% RSLogix 500 project AUTOGENE.RSS, saved by version 8.30.00.16 %
PROJECT "AUTOGENE"    % processor: Bul.1763 MicroLogix 1100 Series B %

PROGRAM FILES
  LAD 2 "MAIN"  4 rungs
  LAD 3 "DIG INPUT"  7 rungs
  LAD 5 "CONTROLS"  6 rungs
  LAD 6 "ALARMS"  12 rungs

DATA FILES
  O0 OUTPUT  6 elements
  I1 INPUT  12 elements
  S2 STATUS  66 elements
  B3 BINARY  4 elements
  T4 TIMER  3 elements
  C5 COUNTER  1 elements
  R6 CONTROL  1 elements
  N7 INTEGER  2 elements
  F8 FLOAT  1 elements

LADDER 2 "MAIN"
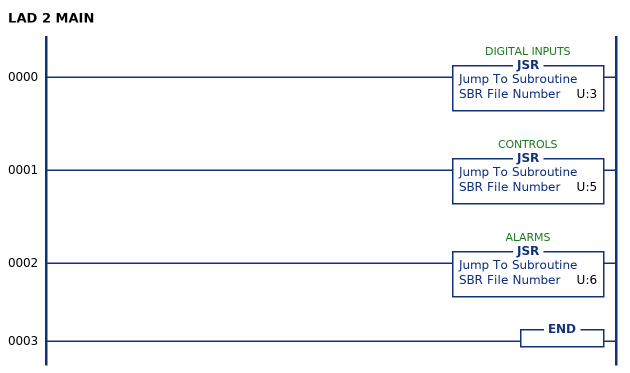
% Rung: 0 %
SOR JSR U:3 EOR
%   U:3  "DIGITAL INPUTS" %
% Rung: 1 %
SOR JSR U:5 EOR
%   U:5  "CONTROLS" %
% Rung: 2 %
SOR JSR U:6 EOR
%   U:6  "ALARMS" %
% Rung: 3 %
SOR END EOR

LADDER 3 "DIG INPUT"
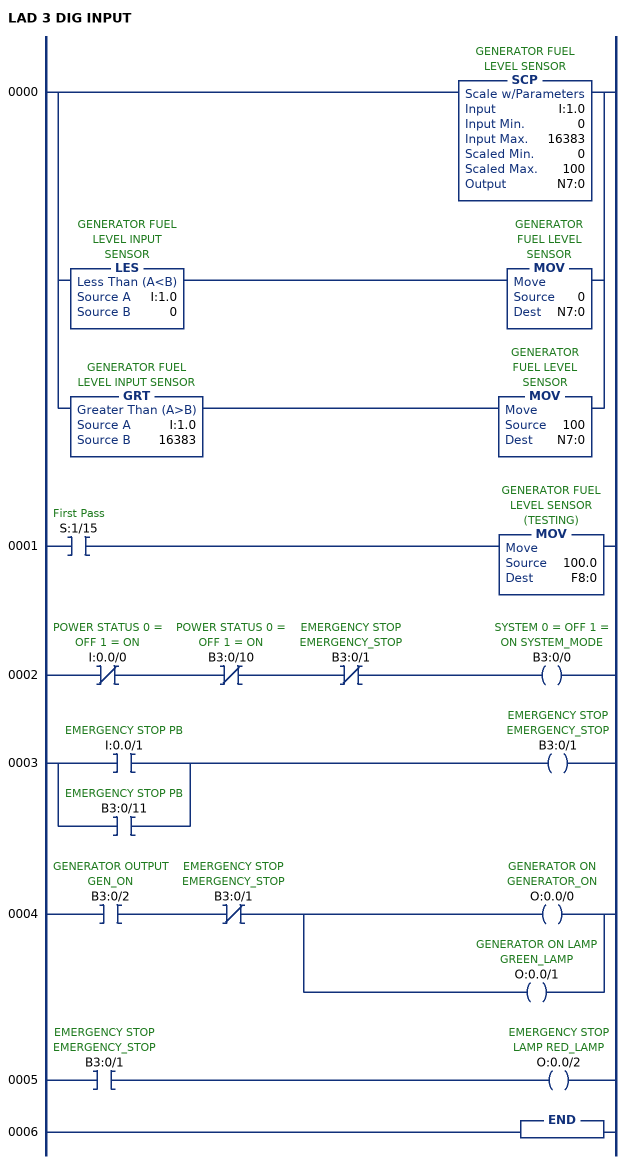
% Rung: 0 %
SOR BST SCP I:1.0 0 16383 0 100 N7:0 NXB LES I:1.0 0 MOV 0 N7:0 NXB GRT I:1.0 16383 MOV 100 N7:0 BND EOR
%   I:1.0  "GENERATOR FUEL LEVEL INPUT SENSOR" %
%   N7:0  "GENERATOR FUEL LEVEL SENSOR" %
% Rung: 1 %
SOR XIC S:1/15 MOV 100.0 F8:0 EOR
%   S:1/15  "First Pass" %
%   F8:0  "GENERATOR FUEL LEVEL SENSOR (TESTING)" %
% Rung: 2 %
SOR XIO I:0.0/0 XIO B3:0/10 XIO B3:0/1 OTE B3:0/0 EOR
%   I:0.0/0  "POWER STATUS 0 = OFF 1 = ON" %
%   B3:0/10  "POWER STATUS 0 = OFF 1 = ON" %
%   B3:0/1  EMERGENCY_STOP  "EMERGENCY STOP" %
%   B3:0/0  SYSTEM_MODE  "SYSTEM 0 = OFF 1 = ON" %
% Rung: 3 %
SOR BST XIC I:0.0/1 NXB XIC B3:0/11 BND OTE B3:0/1 EOR
%   I:0.0/1  "EMERGENCY STOP PB" %
%   B3:0/11  "EMERGENCY STOP PB" %
%   B3:0/1  EMERGENCY_STOP  "EMERGENCY STOP" %
% Rung: 4 %
SOR XIC B3:0/2 XIO B3:0/1 BST OTE O:0.0/0 NXB OTE O:0.0/1 BND EOR
%   B3:0/2  GEN_ON  "GENERATOR OUTPUT" %
%   B3:0/1  EMERGENCY_STOP  "EMERGENCY STOP" %
%   O:0.0/0  GENERATOR_ON  "GENERATOR ON" %
%   O:0.0/1  GREEN_LAMP  "GENERATOR ON LAMP" %
% Rung: 5 %
SOR XIC B3:0/1 OTE O:0.0/2 EOR
%   B3:0/1  EMERGENCY_STOP  "EMERGENCY STOP" %
%   O:0.0/2  RED_LAMP  "EMERGENCY STOP LAMP" %
% Rung: 6 %
SOR END EOR

LADDER 5 "CONTROLS"
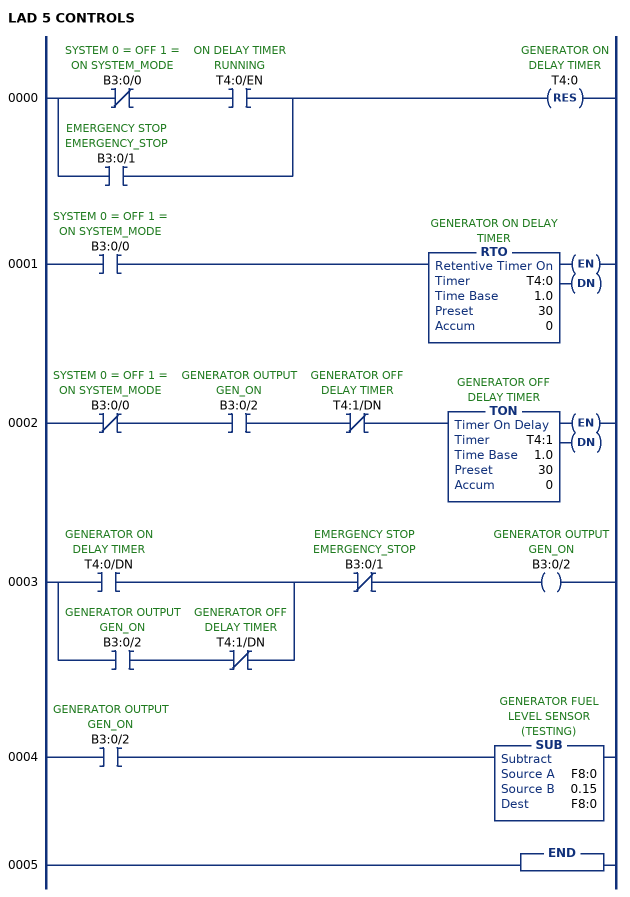
% Rung: 0 %
SOR BST XIO B3:0/0 XIC T4:0/EN NXB XIC B3:0/1 BND RES T4:0 EOR
%   B3:0/0  SYSTEM_MODE  "SYSTEM 0 = OFF 1 = ON" %
%   T4:0/EN  "ON DELAY TIMER RUNNING" %
%   B3:0/1  EMERGENCY_STOP  "EMERGENCY STOP" %
%   T4:0  "GENERATOR ON DELAY TIMER" %
% Rung: 1 %
SOR XIC B3:0/0 RTO T4:0 1.0 30 0 EOR
%   B3:0/0  SYSTEM_MODE  "SYSTEM 0 = OFF 1 = ON" %
%   T4:0  "GENERATOR ON DELAY TIMER" %
% Rung: 2 %
SOR XIO B3:0/0 XIC B3:0/2 XIO T4:1/DN TON T4:1 1.0 30 0 EOR
%   B3:0/0  SYSTEM_MODE  "SYSTEM 0 = OFF 1 = ON" %
%   B3:0/2  GEN_ON  "GENERATOR OUTPUT" %
%   T4:1  "GENERATOR OFF DELAY TIMER" %
% Rung: 3 %
SOR BST XIC T4:0/DN NXB XIC B3:0/2 XIO T4:1/DN BND XIO B3:0/1 OTE B3:0/2 EOR
%   T4:0  "GENERATOR ON DELAY TIMER" %
%   B3:0/2  GEN_ON  "GENERATOR OUTPUT" %
%   T4:1  "GENERATOR OFF DELAY TIMER" %
%   B3:0/1  EMERGENCY_STOP  "EMERGENCY STOP" %
% Rung: 4 %
SOR XIC B3:0/2 SUB F8:0 0.15 F8:0 EOR
%   B3:0/2  GEN_ON  "GENERATOR OUTPUT" %
%   F8:0  "GENERATOR FUEL LEVEL SENSOR (TESTING)" %
% Rung: 5 %
SOR END EOR

LADDER 6 "ALARMS"
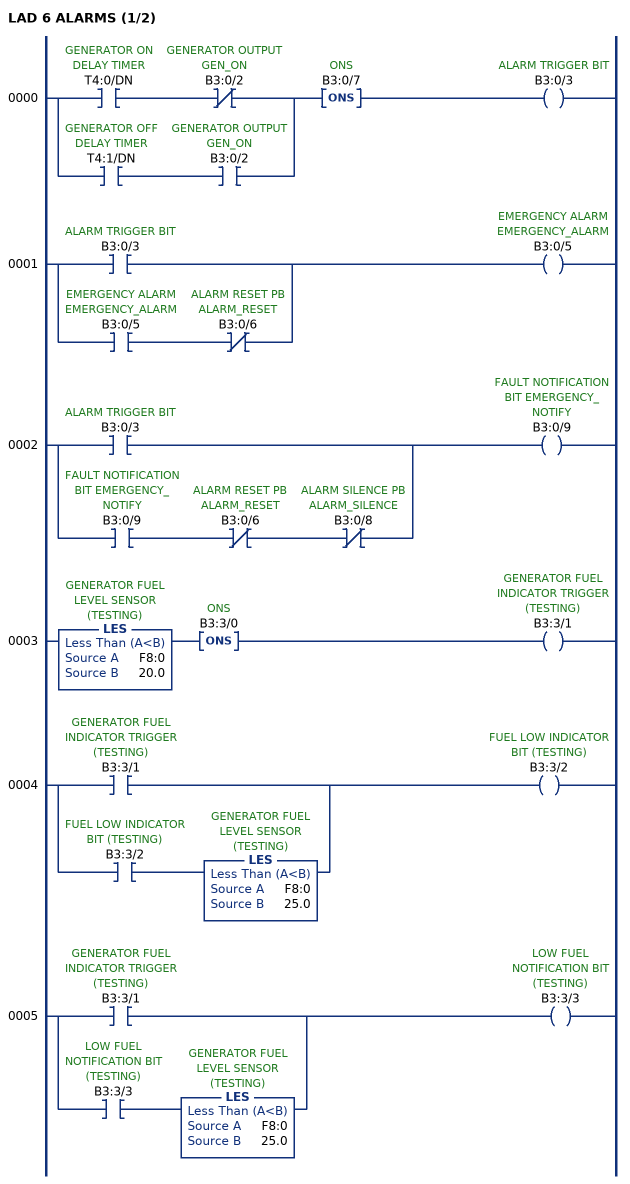
% Rung: 0 %
SOR BST XIC T4:0/DN XIO B3:0/2 NXB XIC T4:1/DN XIC B3:0/2 BND ONS B3:0/7 OTE B3:0/3 EOR
%   T4:0  "GENERATOR ON DELAY TIMER" %
%   B3:0/2  GEN_ON  "GENERATOR OUTPUT" %
%   T4:1  "GENERATOR OFF DELAY TIMER" %
%   B3:0/7  "ONS" %
%   B3:0/3  "ALARM TRIGGER BIT" %
% Rung: 1 %
SOR BST XIC B3:0/3 NXB XIC B3:0/5 XIO B3:0/6 BND OTE B3:0/5 EOR
%   B3:0/3  "ALARM TRIGGER BIT" %
%   B3:0/5  EMERGENCY_ALARM  "EMERGENCY ALARM" %
%   B3:0/6  ALARM_RESET  "ALARM RESET PB" %
% Rung: 2 %
SOR BST XIC B3:0/3 NXB XIC B3:0/9 XIO B3:0/6 XIO B3:0/8 BND OTE B3:0/9 EOR
%   B3:0/3  "ALARM TRIGGER BIT" %
%   B3:0/9  EMERGENCY_NOTIFY  "FAULT NOTIFICATION BIT" %
%   B3:0/6  ALARM_RESET  "ALARM RESET PB" %
%   B3:0/8  ALARM_SILENCE  "ALARM SILENCE PB" %
% Rung: 3 %
SOR LES F8:0 20.0 ONS B3:3/0 OTE B3:3/1 EOR
%   F8:0  "GENERATOR FUEL LEVEL SENSOR (TESTING)" %
%   B3:3/0  "ONS" %
%   B3:3/1  "GENERATOR FUEL INDICATOR TRIGGER (TESTING)" %
% Rung: 4 %
SOR BST XIC B3:3/1 NXB XIC B3:3/2 LES F8:0 25.0 BND OTE B3:3/2 EOR
%   B3:3/1  "GENERATOR FUEL INDICATOR TRIGGER (TESTING)" %
%   B3:3/2  "FUEL LOW INDICATOR BIT (TESTING)" %
%   F8:0  "GENERATOR FUEL LEVEL SENSOR (TESTING)" %
% Rung: 5 %
SOR BST XIC B3:3/1 NXB XIC B3:3/3 LES F8:0 25.0 BND OTE B3:3/3 EOR
%   B3:3/1  "GENERATOR FUEL INDICATOR TRIGGER (TESTING)" %
%   B3:3/3  "LOW FUEL NOTIFICATION BIT (TESTING)" %
%   F8:0  "GENERATOR FUEL LEVEL SENSOR (TESTING)" %

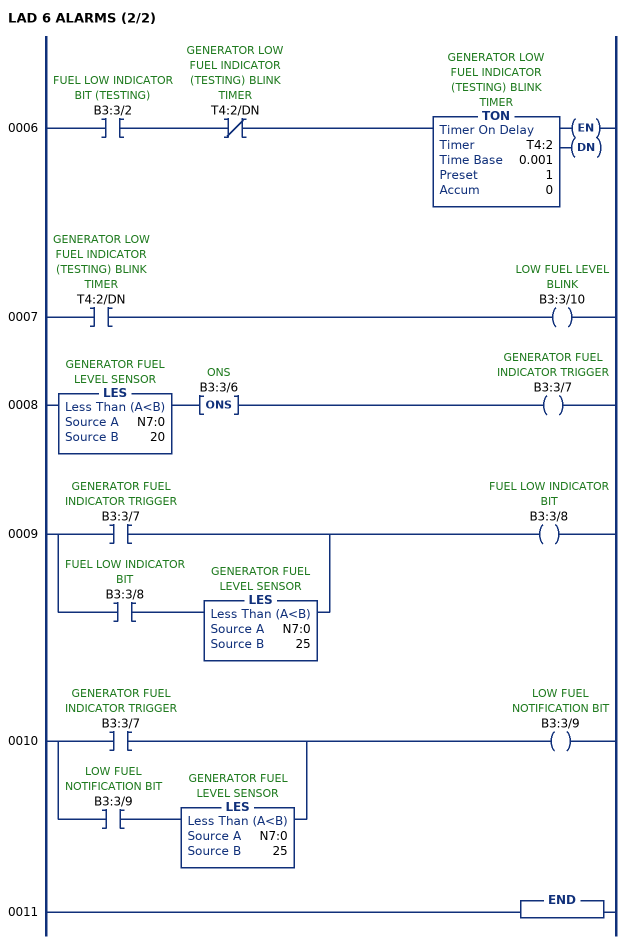
% Rung: 6 %
SOR XIC B3:3/2 XIO T4:2/DN TON T4:2 0.001 1 0 EOR
%   B3:3/2  "FUEL LOW INDICATOR BIT (TESTING)" %
%   T4:2  "GENERATOR LOW FUEL INDICATOR (TESTING) BLINK TIMER" %
% Rung: 7 %
SOR XIC T4:2/DN OTE B3:3/10 EOR
%   T4:2  "GENERATOR LOW FUEL INDICATOR (TESTING) BLINK TIMER" %
%   B3:3/10  "LOW FUEL LEVEL BLINK" %
% Rung: 8 %
SOR LES N7:0 20 ONS B3:3/6 OTE B3:3/7 EOR
%   N7:0  "GENERATOR FUEL LEVEL SENSOR" %
%   B3:3/6  "ONS" %
%   B3:3/7  "GENERATOR FUEL INDICATOR TRIGGER" %
% Rung: 9 %
SOR BST XIC B3:3/7 NXB XIC B3:3/8 LES N7:0 25 BND OTE B3:3/8 EOR
%   B3:3/7  "GENERATOR FUEL INDICATOR TRIGGER" %
%   B3:3/8  "FUEL LOW INDICATOR BIT" %
%   N7:0  "GENERATOR FUEL LEVEL SENSOR" %
% Rung: 10 %
SOR BST XIC B3:3/7 NXB XIC B3:3/9 LES N7:0 25 BND OTE B3:3/9 EOR
%   B3:3/7  "GENERATOR FUEL INDICATOR TRIGGER" %
%   B3:3/9  "LOW FUEL NOTIFICATION BIT" %
%   N7:0  "GENERATOR FUEL LEVEL SENSOR" %
% Rung: 11 %
SOR END EOR

OTHER DOCUMENTED ADDRESSES
  B3:0/4  "ONS"
  B3:1  SYSTEM_ON  "SYS_MODE"
  B3:1/0  "POWER STATUS 0 = OFF 1 = ON"
  B3:2  SYSTEM_OFF  "SYS_MODE"
  B3:2/0  "POWER STATUS 0 = OFF 1 = ON"
  B3:3/4  "ONS"
  B3:3/5  "GENERATOR FUEL LEVEL SENSOR (TESTING) DRAIN TRIGGER"
  I:0.1  "POWER STATUS 0 = OFF 1 = ON"
  I:0.2  "POWER STATUS 0 = OFF 1 = ON"
  N7:1  "GENERATOR FUEL LEVEL SENSOR (TESTING)"
  T4:1/EN  "OFF DELAY TIMER RUNNING"
  U:4  "DIGITAL OUTPUTS"

DATA TABLE (non-zero values as saved)
DATA T4
% .PRE .ACC %
% T4:0 % 30 0
% T4:1 % 30 0
% T4:2 % 1 0
